// TIA Portal V20 export
TYPE "Functional_Test"
   STRUCT
      Water_Fountain : String;
      Serial_Number : String[17];
      Panel_Number : SInt;
      Read_Electrical_Voltage : UInt;
      Read_Electrical_Current : UInt;
      Electrical_Current_Test : String[10];
      Visual_Test : String[10];
      Functional_Test : String[10];
   END_STRUCT;
END_TYPE
